PROGRAM MAIN
VAR
	bInitialise: 		BOOL:= True;
	fbTestsuites:		FB_Testsuites;
	fbTestsuite1:		FB_Testsuite;
	
	fbComponent:		FB_Component;
	
	bReset:			BOOL;
	bStart: 		BOOL;
    bHold:       	BOOL;
    bPause:    		BOOL;
	bStop:       	BOOL;
    bAbort:      	BOOL;

	bExecute: BOOL;
END_VAR

IF bInitialise THEN
	bInitialise:= False;
	fbTestsuites.M_Add(fbTestsuite1);
	fbTestsuites.P_Options.sFilePathName:= 'C:\report.xml';
	fbTestsuite1.P_Options.bAbortOnError:= FALSE;
END_IF

IF bExecute THEN
	bExecute:= fbTestsuites.M_Request(E_Base.Execute);
END_IF

fbTestsuites();
fbTestsuite1();

fbComponent.M_Cycle();

CASE fbTestsuite1.P_Testcase OF
	
	E_Testcase.Start:
		fbTestsuite1.P_Assert.M_Equals_BOOL(TRUE, fbComponent.M_Request(E_Request.Reset), 'Reset');
		fbTestsuite1.P_Assert.M_Equals_INT(E_State.Idle, fbComponent.P_State, 'E_State.Idle');
		fbTestsuite1.M_Testcase('FB_Component', T#1S, 'fbComponent.M_Request(E_Request.Reset)', '', 10);	
	
	10:	
		fbTestsuite1.P_Assert.M_Equals_BOOL(TRUE, fbComponent.M_Request(E_Request.Start), 'Start');
		fbTestsuite1.P_Assert.M_Equals_INT(E_State.Execute, fbComponent.P_State, 'E_State.Execute');
		fbTestsuite1.M_Testcase('FB_Component', T#1S, 'fbComponent.M_Request(E_Request.Start)', '', 20);
		
	20:
		fbTestsuite1.P_Assert.M_Equals_BOOL(TRUE, fbComponent.M_Request(E_Request.Stop), 'Stop');
		fbTestsuite1.P_Assert.M_Equals_INT(E_State.Stopped, fbComponent.P_State, 'E_State.Stop');
		fbTestsuite1.M_Testcase('FB_Component', T#1S, 'fbComponent.M_Request(E_Request.Stop)', '', 30);
		
	30:
		fbTestsuite1.P_Assert.M_Equals_BOOL(TRUE, fbComponent.M_Request(E_Request.Reset), 'Reset');
		fbTestsuite1.P_Assert.M_Equals_INT(E_State.Idle, fbComponent.P_State, 'E_State.Idle');
		fbTestsuite1.M_Testcase('FB_Component', T#1S, 'fbComponent.M_Request(E_Request.Reset)', '', 40);
		
	40:	
		fbTestsuite1.P_Assert.M_Equals_BOOL(TRUE, fbComponent.M_Request(E_Request.Start), 'Start');
		fbTestsuite1.P_Assert.M_Equals_INT(E_State.Execute, fbComponent.P_State, 'E_State.Execute');
		fbTestsuite1.M_Testcase('FB_Component', T#1S, 'fbComponent.M_Request(E_Request.Start)', '', 50);
		
	50:	
		fbTestsuite1.P_Assert.M_Equals_BOOL(TRUE, fbComponent.M_Request(E_Request.Abort), 'Abort');
		fbTestsuite1.P_Assert.M_Equals_INT(E_State.Aborted, fbComponent.P_State, 'E_State.Aborted');
		fbTestsuite1.M_Testcase('FB_Component', T#1S, 'fbComponent.M_Request(E_Request.Abort)', '', 60);
		
	60:
		fbTestsuite1.P_Assert.M_Equals_BOOL(TRUE, fbComponent.M_Request(E_Request.Reset), 'Reset');
		fbTestsuite1.P_Assert.M_Equals_INT(E_State.Idle, fbComponent.P_State, 'E_State.Idle');
		fbTestsuite1.M_Testcase('FB_Component', T#1S, 'fbComponent.M_Request(E_Request.Reset)', '', 70);
		
	70:	
		fbTestsuite1.P_Assert.M_Equals_BOOL(TRUE, fbComponent.M_Request(E_Request.Start), 'Start');
		fbTestsuite1.P_Assert.M_Equals_INT(E_State.Execute, fbComponent.P_State, 'E_State.Execute');
		fbTestsuite1.M_Testcase('FB_Component', T#1S, 'fbComponent.M_Request(E_Request.Start)', '', 80);	
	
	80:	
		fbTestsuite1.P_Assert.M_Equals_BOOL(TRUE, fbComponent.M_Request(E_Request.Complete), 'Complete');
		fbTestsuite1.P_Assert.M_Equals_INT(E_State.Completed, fbComponent.P_State, 'E_State.Execute');
		fbTestsuite1.M_Testcase('FB_Component', T#1S, 'fbComponent.M_Request(E_Request.Complete)', '', 90);		

	90:
		fbTestsuite1.P_Assert.M_Equals_BOOL(TRUE, fbComponent.M_Request(E_Request.Reset), 'Reset');
		fbTestsuite1.P_Assert.M_Equals_INT(E_State.Idle, fbComponent.P_State, 'E_State.Idle');
		fbTestsuite1.M_Testcase('FB_Component', T#1S, 'fbComponent.M_Request(E_Request.Reset)', '', E_Testcase.Done);		
		
	E_Testcase.Done:;
	
END_CASE

END_PROGRAM

(* stored: Version 1.1.0.1
   POU MAIN: Id {4321fa7e-09fb-4f02-847a-cf67275926df}, SpecialFunc None *)
